Staubli VAL3: moveDown.pgx

program moveDown(pointRs where, mdesc finalSpeed, trsf finalAppro, bool meticulous, trsf xyTrsf)
  local mdesc speed[3]
begin
  // Note: finalSpeed is not taken literally!
  if finalSpeed == mVerySlow
    speed[0] = mFast
    speed[1] = mSlow
    speed[2] = mVerySlow
  elseIf finalSpeed == mSlow
    speed[0] = mFast
    speed[1] = mSlow
    speed[2] = mSlow
  else
    speed[0] = mFast
    speed[1] = mFast
    speed[2] = mSlow
  endIf

  //movej(appro(where, trZsafe*xyTrsf), tTool, speed[0])
  movej(appro(where, trZsafe), tTool, speed[0])
  if meticulous
    waitEndMove()
  endIf

  // -- move down with decreasing speeds. Not sure whether this gets "blended" away
  //movej(appro(where, trZclose*xyTrsf), tTool, speed[1])
  //movej(appro(where, finalAppro*xyTrsf), tTool, speed[2])

  movej(appro(where, trZclose), tTool, speed[1])
  movej(appro(where, finalAppro), tTool, speed[2])
  waitEndMove()
end
